// TIA Portal V20 export
TYPE "LER_typeGearInControlNodes"
// stored: Access Published
   STRUCT
      command : "LER_typeGearInCommand";
      monitoring : "LER_typeGearInMonitoring";
   END_STRUCT;
END_TYPE
